// TIA Portal V20 export
ORGANIZATION_BLOCK "Main"   // OB1, LAD, ProgramCycle
TITLE = "Main Program Sweep (Cycle)"
{ S7_Optimized_Access := 'TRUE' }
// stored: SetENOAutomatically false
   VAR_INPUT
      Initial_Call : Bool;   // Initial call of this OB
      Remanence : Bool;   // =True, if remanent data are available
   END_VAR
BEGIN

REGION Network 1: SideShifter2
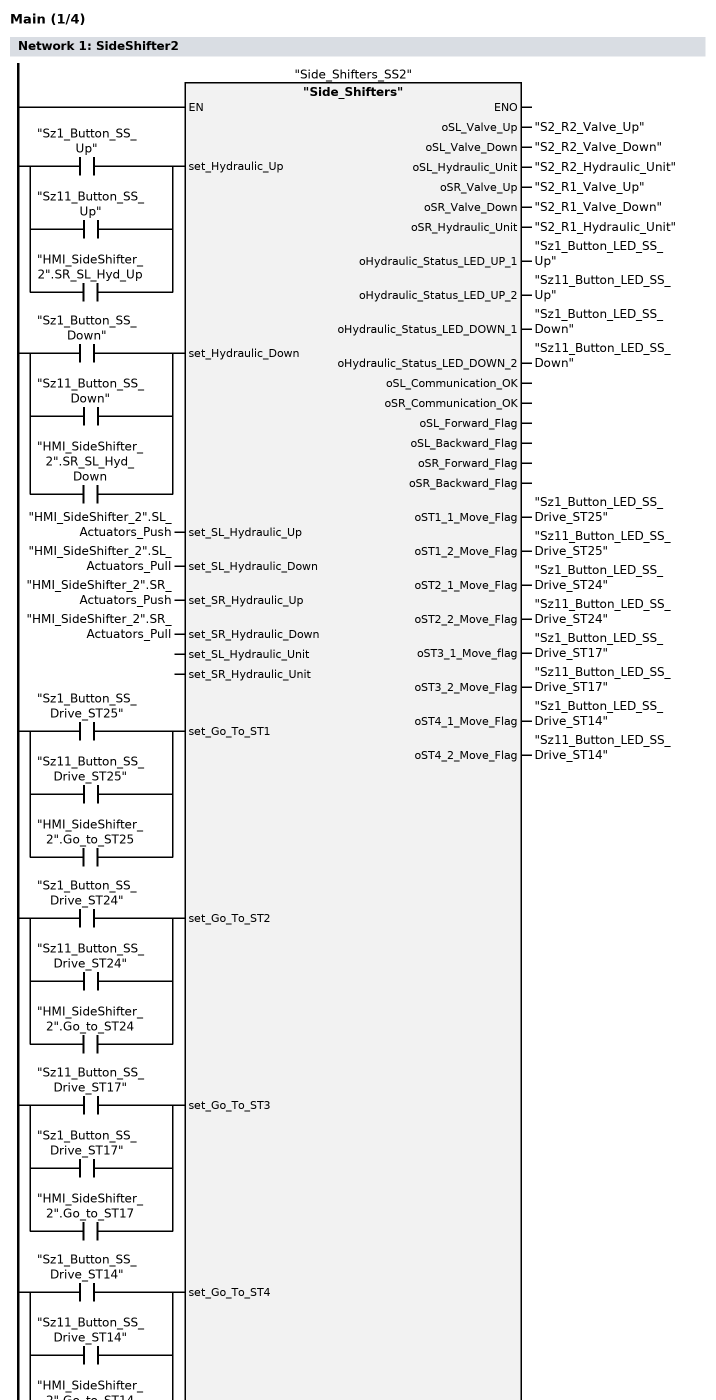
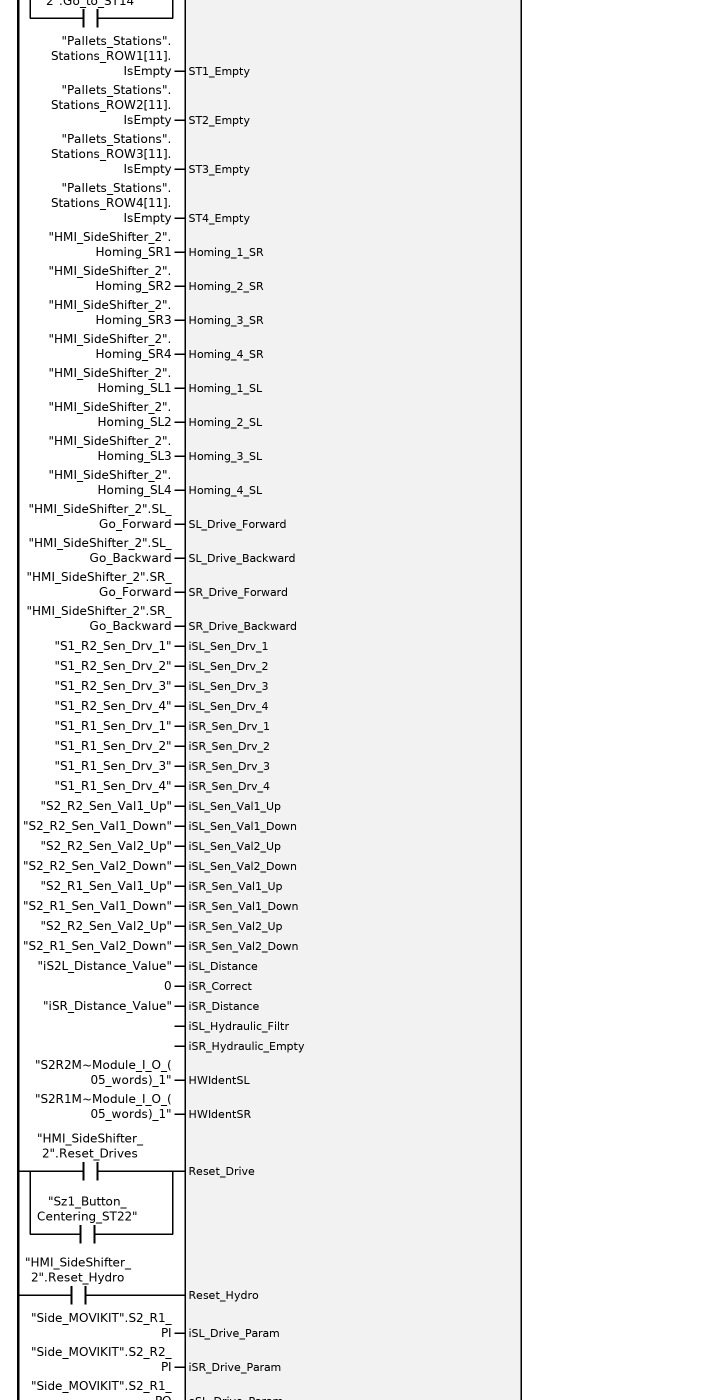
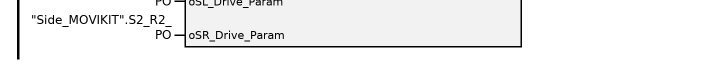
   RUNG wire#powerrail
      "Side_Shifters_SS2"(set_Hydraulic_Up := wire#w1, set_Hydraulic_Down := wire#w2, set_Go_To_ST1 := wire#w3, set_Go_To_ST2 := wire#w4, set_Go_To_ST3 := wire#w5, set_Go_To_ST4 := wire#w6, Reset_Drive := wire#w7, Reset_Hydro := wire#w8, set_SL_Hydraulic_Up := "HMI_SideShifter_2".SL_Actuators_Push, set_SL_Hydraulic_Down := "HMI_SideShifter_2".SL_Actuators_Pull, set_SR_Hydraulic_Up := "HMI_SideShifter_2".SR_Actuators_Push, set_SR_Hydraulic_Down := "HMI_SideShifter_2".SR_Actuators_Pull, set_SL_Hydraulic_Unit :=, set_SR_Hydraulic_Unit :=, ST1_Empty := "Pallets_Stations".Stations_ROW1[11].IsEmpty, ST2_Empty := "Pallets_Stations".Stations_ROW2[11].IsEmpty, ST3_Empty := "Pallets_Stations".Stations_ROW3[11].IsEmpty, ST4_Empty := "Pallets_Stations".Stations_ROW4[11].IsEmpty, Homing_1_SR := "HMI_SideShifter_2".Homing_SR1, Homing_2_SR := "HMI_SideShifter_2".Homing_SR2, Homing_3_SR := "HMI_SideShifter_2".Homing_SR3, Homing_4_SR := "HMI_SideShifter_2".Homing_SR4, Homing_1_SL := "HMI_SideShifter_2".Homing_SL1, Homing_2_SL := "HMI_SideShifter_2".Homing_SL2, Homing_3_SL := "HMI_SideShifter_2".Homing_SL3, Homing_4_SL := "HMI_SideShifter_2".Homing_SL4, SL_Drive_Forward := "HMI_SideShifter_2".SL_Go_Forward, SL_Drive_Backward := "HMI_SideShifter_2".SL_Go_Backward, SR_Drive_Forward := "HMI_SideShifter_2".SR_Go_Forward, SR_Drive_Backward := "HMI_SideShifter_2".SR_Go_Backward, iSL_Sen_Drv_1 := "S1_R2_Sen_Drv_1", iSL_Sen_Drv_2 := "S1_R2_Sen_Drv_2", iSL_Sen_Drv_3 := "S1_R2_Sen_Drv_3", iSL_Sen_Drv_4 := "S1_R2_Sen_Drv_4", iSR_Sen_Drv_1 := "S1_R1_Sen_Drv_1", iSR_Sen_Drv_2 := "S1_R1_Sen_Drv_2", iSR_Sen_Drv_3 := "S1_R1_Sen_Drv_3", iSR_Sen_Drv_4 := "S1_R1_Sen_Drv_4", iSL_Sen_Val1_Up := "S2_R2_Sen_Val1_Up", iSL_Sen_Val1_Down := "S2_R2_Sen_Val1_Down", iSL_Sen_Val2_Up := "S2_R2_Sen_Val2_Up", iSL_Sen_Val2_Down := "S2_R2_Sen_Val2_Down", iSR_Sen_Val1_Up := "S2_R1_Sen_Val1_Up", iSR_Sen_Val1_Down := "S2_R1_Sen_Val1_Down", iSR_Sen_Val2_Up := "S2_R2_Sen_Val2_Up", iSR_Sen_Val2_Down := "S2_R1_Sen_Val2_Down", iSL_Distance := "iS2L_Distance_Value", iSR_Correct := 0, iSR_Distance := "iSR_Distance_Value", iSL_Hydraulic_Filtr :=, iSR_Hydraulic_Empty :=, HWIdentSL := "S2R2M~Module_I_O_(05_words)_1", HWIdentSR := "S2R1M~Module_I_O_(05_words)_1", iSL_Drive_Param := "Side_MOVIKIT".S2_R1_PI, iSR_Drive_Param := "Side_MOVIKIT".S2_R2_PI, oSL_Drive_Param := "Side_MOVIKIT".S2_R1_PO, oSR_Drive_Param := "Side_MOVIKIT".S2_R2_PO, oSL_Valve_Up => "S2_R2_Valve_Up", oSL_Valve_Down => "S2_R2_Valve_Down", oSL_Hydraulic_Unit => "S2_R2_Hydraulic_Unit", oSR_Valve_Up => "S2_R1_Valve_Up", oSR_Valve_Down => "S2_R1_Valve_Down", oSR_Hydraulic_Unit => "S2_R1_Hydraulic_Unit", oHydraulic_Status_LED_UP_1 => "Sz1_Button_LED_SS_Up", oHydraulic_Status_LED_UP_2 => "Sz11_Button_LED_SS_Up", oHydraulic_Status_LED_DOWN_1 => "Sz1_Button_LED_SS_Down", oHydraulic_Status_LED_DOWN_2 => "Sz11_Button_LED_SS_Down", oSL_Communication_OK =>, oSR_Communication_OK =>, oSL_Forward_Flag =>, oSL_Backward_Flag =>, oSR_Forward_Flag =>, oSR_Backward_Flag =>, oST1_1_Move_Flag => "Sz1_Button_LED_SS_Drive_ST25", oST1_2_Move_Flag => "Sz11_Button_LED_SS_Drive_ST25", oST2_1_Move_Flag => "Sz1_Button_LED_SS_Drive_ST24", oST2_2_Move_Flag => "Sz11_Button_LED_SS_Drive_ST24", oST3_1_Move_flag => "Sz1_Button_LED_SS_Drive_ST17", oST3_2_Move_Flag => "Sz11_Button_LED_SS_Drive_ST17", oST4_1_Move_Flag => "Sz1_Button_LED_SS_Drive_ST14", oST4_2_Move_Flag => "Sz11_Button_LED_SS_Drive_ST14")
   END_RUNG
   RUNG wire#powerrail
      Contact( "Sz1_Button_SS_Up" )
   END_RUNG wire#w1
   RUNG wire#powerrail
      Contact( "Sz11_Button_SS_Up" )
   END_RUNG wire#w1
   RUNG wire#powerrail
      Contact( "HMI_SideShifter_2".SR_SL_Hyd_Up )
   END_RUNG wire#w1
   RUNG wire#powerrail
      Contact( "Sz1_Button_SS_Down" )
   END_RUNG wire#w2
   RUNG wire#powerrail
      Contact( "Sz11_Button_SS_Down" )
   END_RUNG wire#w2
   RUNG wire#powerrail
      Contact( "HMI_SideShifter_2".SR_SL_Hyd_Down )
   END_RUNG wire#w2
   RUNG wire#powerrail
      Contact( "Sz1_Button_SS_Drive_ST25" )
   END_RUNG wire#w3
   RUNG wire#powerrail
      Contact( "Sz11_Button_SS_Drive_ST25" )
   END_RUNG wire#w3
   RUNG wire#powerrail
      Contact( "HMI_SideShifter_2".Go_to_ST25 )
   END_RUNG wire#w3
   RUNG wire#powerrail
      Contact( "Sz1_Button_SS_Drive_ST24" )
   END_RUNG wire#w4
   RUNG wire#powerrail
      Contact( "Sz11_Button_SS_Drive_ST24" )
   END_RUNG wire#w4
   RUNG wire#powerrail
      Contact( "HMI_SideShifter_2".Go_to_ST24 )
   END_RUNG wire#w4
   RUNG wire#powerrail
      Contact( "Sz11_Button_SS_Drive_ST17" )
   END_RUNG wire#w5
   RUNG wire#powerrail
      Contact( "Sz1_Button_SS_Drive_ST17" )
   END_RUNG wire#w5
   RUNG wire#powerrail
      Contact( "HMI_SideShifter_2".Go_to_ST17 )
   END_RUNG wire#w5
   RUNG wire#powerrail
      Contact( "Sz1_Button_SS_Drive_ST14" )
   END_RUNG wire#w6
   RUNG wire#powerrail
      Contact( "Sz11_Button_SS_Drive_ST14" )
   END_RUNG wire#w6
   RUNG wire#powerrail
      Contact( "HMI_SideShifter_2".Go_to_ST14 )
   END_RUNG wire#w6
   RUNG wire#powerrail
      Contact( "HMI_SideShifter_2".Reset_Drives )
   END_RUNG wire#w7
   RUNG wire#powerrail
      Contact( "Sz1_Button_Centering_ST22" )
   END_RUNG wire#w7
   RUNG wire#powerrail
      Contact( "HMI_SideShifter_2".Reset_Hydro )
   END_RUNG wire#w8
   // the same network as SCL:
   "Side_Shifters_SS2"(set_Hydraulic_Up := "Sz1_Button_SS_Up" OR "Sz11_Button_SS_Up" OR "HMI_SideShifter_2".SR_SL_Hyd_Up,   // "Side_Shifters"
                       set_Hydraulic_Down := "Sz1_Button_SS_Down" OR "Sz11_Button_SS_Down" OR "HMI_SideShifter_2".SR_SL_Hyd_Down,
                       set_SL_Hydraulic_Up := "HMI_SideShifter_2".SL_Actuators_Push,
                       set_SL_Hydraulic_Down := "HMI_SideShifter_2".SL_Actuators_Pull,
                       set_SR_Hydraulic_Up := "HMI_SideShifter_2".SR_Actuators_Push,
                       set_SR_Hydraulic_Down := "HMI_SideShifter_2".SR_Actuators_Pull,
                       set_Go_To_ST1 := "Sz1_Button_SS_Drive_ST25" OR "Sz11_Button_SS_Drive_ST25" OR "HMI_SideShifter_2".Go_to_ST25,
                       set_Go_To_ST2 := "Sz1_Button_SS_Drive_ST24" OR "Sz11_Button_SS_Drive_ST24" OR "HMI_SideShifter_2".Go_to_ST24,
                       set_Go_To_ST3 := "Sz11_Button_SS_Drive_ST17" OR "Sz1_Button_SS_Drive_ST17" OR "HMI_SideShifter_2".Go_to_ST17,
                       set_Go_To_ST4 := "Sz1_Button_SS_Drive_ST14" OR "Sz11_Button_SS_Drive_ST14" OR "HMI_SideShifter_2".Go_to_ST14,
                       ST1_Empty := "Pallets_Stations".Stations_ROW1[11].IsEmpty,
                       ST2_Empty := "Pallets_Stations".Stations_ROW2[11].IsEmpty,
                       ST3_Empty := "Pallets_Stations".Stations_ROW3[11].IsEmpty,
                       ST4_Empty := "Pallets_Stations".Stations_ROW4[11].IsEmpty,
                       Homing_1_SR := "HMI_SideShifter_2".Homing_SR1,
                       Homing_2_SR := "HMI_SideShifter_2".Homing_SR2,
                       Homing_3_SR := "HMI_SideShifter_2".Homing_SR3,
                       Homing_4_SR := "HMI_SideShifter_2".Homing_SR4,
                       Homing_1_SL := "HMI_SideShifter_2".Homing_SL1,
                       Homing_2_SL := "HMI_SideShifter_2".Homing_SL2,
                       Homing_3_SL := "HMI_SideShifter_2".Homing_SL3,
                       Homing_4_SL := "HMI_SideShifter_2".Homing_SL4,
                       SL_Drive_Forward := "HMI_SideShifter_2".SL_Go_Forward,
                       SL_Drive_Backward := "HMI_SideShifter_2".SL_Go_Backward,
                       SR_Drive_Forward := "HMI_SideShifter_2".SR_Go_Forward,
                       SR_Drive_Backward := "HMI_SideShifter_2".SR_Go_Backward,
                       iSL_Sen_Drv_1 := "S1_R2_Sen_Drv_1",
                       iSL_Sen_Drv_2 := "S1_R2_Sen_Drv_2",
                       iSL_Sen_Drv_3 := "S1_R2_Sen_Drv_3",
                       iSL_Sen_Drv_4 := "S1_R2_Sen_Drv_4",
                       iSR_Sen_Drv_1 := "S1_R1_Sen_Drv_1",
                       iSR_Sen_Drv_2 := "S1_R1_Sen_Drv_2",
                       iSR_Sen_Drv_3 := "S1_R1_Sen_Drv_3",
                       iSR_Sen_Drv_4 := "S1_R1_Sen_Drv_4",
                       iSL_Sen_Val1_Up := "S2_R2_Sen_Val1_Up",
                       iSL_Sen_Val1_Down := "S2_R2_Sen_Val1_Down",
                       iSL_Sen_Val2_Up := "S2_R2_Sen_Val2_Up",
                       iSL_Sen_Val2_Down := "S2_R2_Sen_Val2_Down",
                       iSR_Sen_Val1_Up := "S2_R1_Sen_Val1_Up",
                       iSR_Sen_Val1_Down := "S2_R1_Sen_Val1_Down",
                       iSR_Sen_Val2_Up := "S2_R2_Sen_Val2_Up",
                       iSR_Sen_Val2_Down := "S2_R1_Sen_Val2_Down",
                       iSL_Distance := "iS2L_Distance_Value",
                       iSR_Correct := 0,
                       iSR_Distance := "iSR_Distance_Value",
                       HWIdentSL := "S2R2M~Module_I_O_(05_words)_1",
                       HWIdentSR := "S2R1M~Module_I_O_(05_words)_1",
                       Reset_Drive := "HMI_SideShifter_2".Reset_Drives OR "Sz1_Button_Centering_ST22",
                       Reset_Hydro := "HMI_SideShifter_2".Reset_Hydro,
                       iSL_Drive_Param := "Side_MOVIKIT".S2_R1_PI,
                       iSR_Drive_Param := "Side_MOVIKIT".S2_R2_PI,
                       oSL_Drive_Param := "Side_MOVIKIT".S2_R1_PO,
                       oSR_Drive_Param := "Side_MOVIKIT".S2_R2_PO,
                       oSL_Valve_Up => "S2_R2_Valve_Up",
                       oSL_Valve_Down => "S2_R2_Valve_Down",
                       oSL_Hydraulic_Unit => "S2_R2_Hydraulic_Unit",
                       oSR_Valve_Up => "S2_R1_Valve_Up",
                       oSR_Valve_Down => "S2_R1_Valve_Down",
                       oSR_Hydraulic_Unit => "S2_R1_Hydraulic_Unit",
                       oHydraulic_Status_LED_UP_1 => "Sz1_Button_LED_SS_Up",
                       oHydraulic_Status_LED_UP_2 => "Sz11_Button_LED_SS_Up",
                       oHydraulic_Status_LED_DOWN_1 => "Sz1_Button_LED_SS_Down",
                       oHydraulic_Status_LED_DOWN_2 => "Sz11_Button_LED_SS_Down",
                       oST1_1_Move_Flag => "Sz1_Button_LED_SS_Drive_ST25",
                       oST1_2_Move_Flag => "Sz11_Button_LED_SS_Drive_ST25",
                       oST2_1_Move_Flag => "Sz1_Button_LED_SS_Drive_ST24",
                       oST2_2_Move_Flag => "Sz11_Button_LED_SS_Drive_ST24",
                       oST3_1_Move_flag => "Sz1_Button_LED_SS_Drive_ST17",
                       oST3_2_Move_Flag => "Sz11_Button_LED_SS_Drive_ST17",
                       oST4_1_Move_Flag => "Sz1_Button_LED_SS_Drive_ST14",
                       oST4_2_Move_Flag => "Sz11_Button_LED_SS_Drive_ST14");
END_REGION

REGION Network 2: SideShifter 1
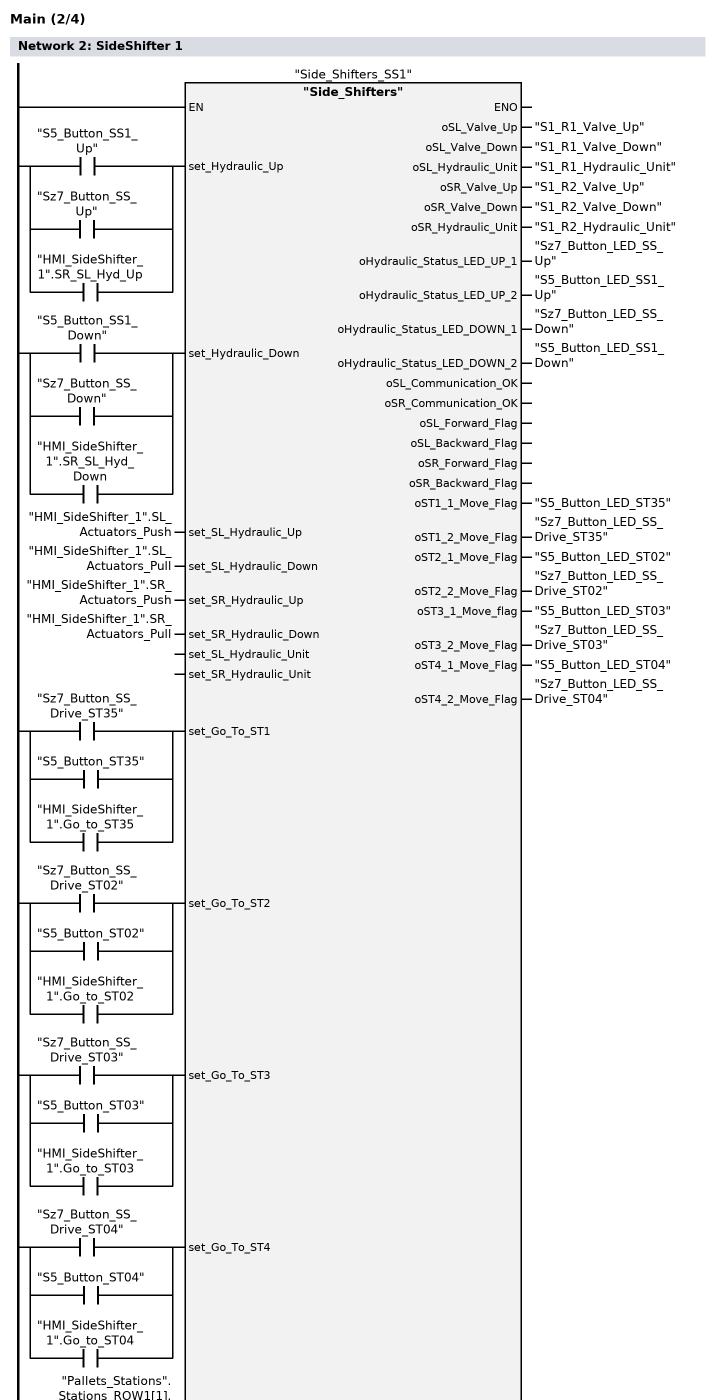
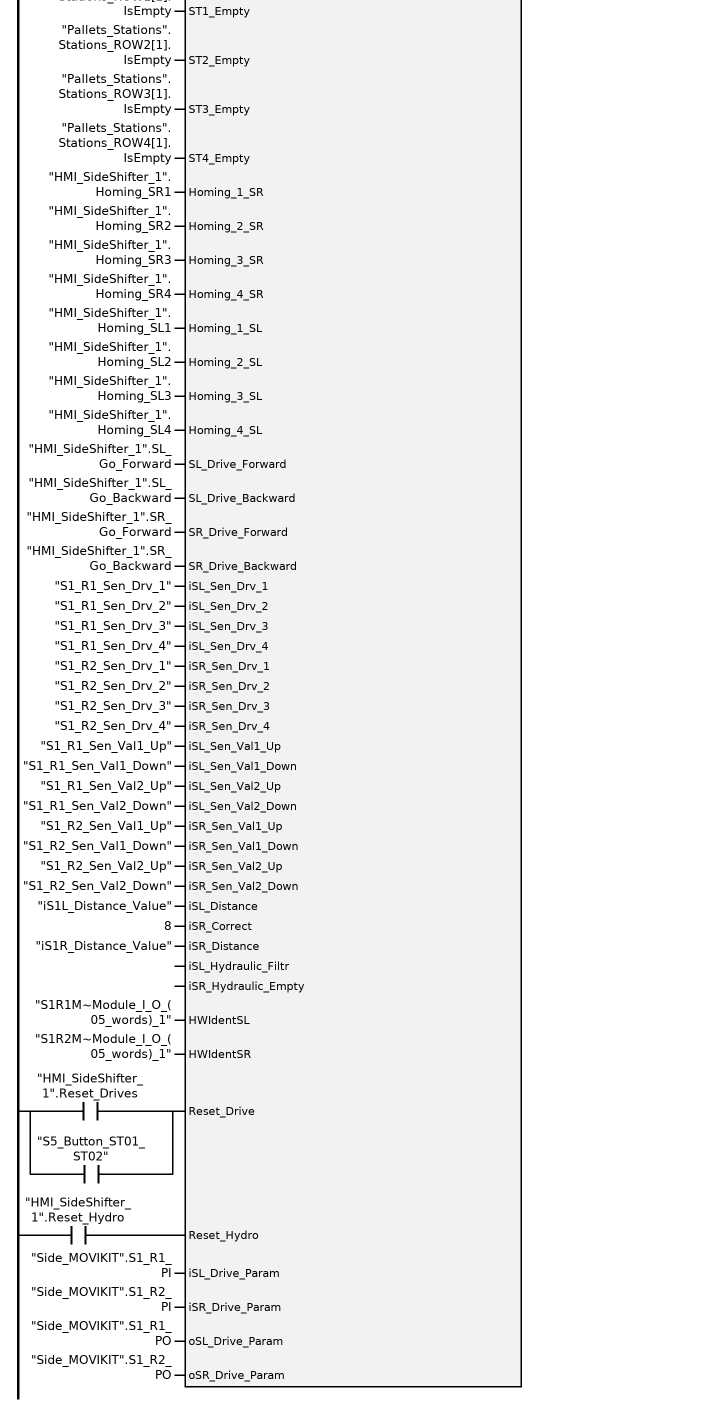
   RUNG wire#powerrail
      "Side_Shifters_SS1"(set_Hydraulic_Up := wire#w1, set_Hydraulic_Down := wire#w2, set_Go_To_ST1 := wire#w3, set_Go_To_ST2 := wire#w4, set_Go_To_ST3 := wire#w5, set_Go_To_ST4 := wire#w6, Reset_Drive := wire#w7, Reset_Hydro := wire#w8, set_SL_Hydraulic_Up := "HMI_SideShifter_1".SL_Actuators_Push, set_SL_Hydraulic_Down := "HMI_SideShifter_1".SL_Actuators_Pull, set_SR_Hydraulic_Up := "HMI_SideShifter_1".SR_Actuators_Push, set_SR_Hydraulic_Down := "HMI_SideShifter_1".SR_Actuators_Pull, set_SL_Hydraulic_Unit :=, set_SR_Hydraulic_Unit :=, ST1_Empty := "Pallets_Stations".Stations_ROW1[1].IsEmpty, ST2_Empty := "Pallets_Stations".Stations_ROW2[1].IsEmpty, ST3_Empty := "Pallets_Stations".Stations_ROW3[1].IsEmpty, ST4_Empty := "Pallets_Stations".Stations_ROW4[1].IsEmpty, Homing_1_SR := "HMI_SideShifter_1".Homing_SR1, Homing_2_SR := "HMI_SideShifter_1".Homing_SR2, Homing_3_SR := "HMI_SideShifter_1".Homing_SR3, Homing_4_SR := "HMI_SideShifter_1".Homing_SR4, Homing_1_SL := "HMI_SideShifter_1".Homing_SL1, Homing_2_SL := "HMI_SideShifter_1".Homing_SL2, Homing_3_SL := "HMI_SideShifter_1".Homing_SL3, Homing_4_SL := "HMI_SideShifter_1".Homing_SL4, SL_Drive_Forward := "HMI_SideShifter_1".SL_Go_Forward, SL_Drive_Backward := "HMI_SideShifter_1".SL_Go_Backward, SR_Drive_Forward := "HMI_SideShifter_1".SR_Go_Forward, SR_Drive_Backward := "HMI_SideShifter_1".SR_Go_Backward, iSL_Sen_Drv_1 := "S1_R1_Sen_Drv_1", iSL_Sen_Drv_2 := "S1_R1_Sen_Drv_2", iSL_Sen_Drv_3 := "S1_R1_Sen_Drv_3", iSL_Sen_Drv_4 := "S1_R1_Sen_Drv_4", iSR_Sen_Drv_1 := "S1_R2_Sen_Drv_1", iSR_Sen_Drv_2 := "S1_R2_Sen_Drv_2", iSR_Sen_Drv_3 := "S1_R2_Sen_Drv_3", iSR_Sen_Drv_4 := "S1_R2_Sen_Drv_4", iSL_Sen_Val1_Up := "S1_R1_Sen_Val1_Up", iSL_Sen_Val1_Down := "S1_R1_Sen_Val1_Down", iSL_Sen_Val2_Up := "S1_R1_Sen_Val2_Up", iSL_Sen_Val2_Down := "S1_R1_Sen_Val2_Down", iSR_Sen_Val1_Up := "S1_R2_Sen_Val1_Up", iSR_Sen_Val1_Down := "S1_R2_Sen_Val1_Down", iSR_Sen_Val2_Up := "S1_R2_Sen_Val2_Up", iSR_Sen_Val2_Down := "S1_R2_Sen_Val2_Down", iSL_Distance := "iS1L_Distance_Value", iSR_Correct := 8, iSR_Distance := "iS1R_Distance_Value", iSL_Hydraulic_Filtr :=, iSR_Hydraulic_Empty :=, HWIdentSL := "S1R1M~Module_I_O_(05_words)_1", HWIdentSR := "S1R2M~Module_I_O_(05_words)_1", iSL_Drive_Param := "Side_MOVIKIT".S1_R1_PI, iSR_Drive_Param := "Side_MOVIKIT".S1_R2_PI, oSL_Drive_Param := "Side_MOVIKIT".S1_R1_PO, oSR_Drive_Param := "Side_MOVIKIT".S1_R2_PO, oSL_Valve_Up => "S1_R1_Valve_Up", oSL_Valve_Down => "S1_R1_Valve_Down", oSL_Hydraulic_Unit => "S1_R1_Hydraulic_Unit", oSR_Valve_Up => "S1_R2_Valve_Up", oSR_Valve_Down => "S1_R2_Valve_Down", oSR_Hydraulic_Unit => "S1_R2_Hydraulic_Unit", oHydraulic_Status_LED_UP_1 => "Sz7_Button_LED_SS_Up", oHydraulic_Status_LED_UP_2 => "S5_Button_LED_SS1_Up", oHydraulic_Status_LED_DOWN_1 => "Sz7_Button_LED_SS_Down", oHydraulic_Status_LED_DOWN_2 => "S5_Button_LED_SS1_Down", oSL_Communication_OK =>, oSR_Communication_OK =>, oSL_Forward_Flag =>, oSL_Backward_Flag =>, oSR_Forward_Flag =>, oSR_Backward_Flag =>, oST1_1_Move_Flag => "S5_Button_LED_ST35", oST1_2_Move_Flag => "Sz7_Button_LED_SS_Drive_ST35", oST2_1_Move_Flag => "S5_Button_LED_ST02", oST2_2_Move_Flag => "Sz7_Button_LED_SS_Drive_ST02", oST3_1_Move_flag => "S5_Button_LED_ST03", oST3_2_Move_Flag => "Sz7_Button_LED_SS_Drive_ST03", oST4_1_Move_Flag => "S5_Button_LED_ST04", oST4_2_Move_Flag => "Sz7_Button_LED_SS_Drive_ST04")
   END_RUNG
   RUNG wire#powerrail
      Contact( "S5_Button_SS1_Up" )
   END_RUNG wire#w1
   RUNG wire#powerrail
      Contact( "Sz7_Button_SS_Up" )
   END_RUNG wire#w1
   RUNG wire#powerrail
      Contact( "HMI_SideShifter_1".SR_SL_Hyd_Up )
   END_RUNG wire#w1
   RUNG wire#powerrail
      Contact( "S5_Button_SS1_Down" )
   END_RUNG wire#w2
   RUNG wire#powerrail
      Contact( "Sz7_Button_SS_Down" )
   END_RUNG wire#w2
   RUNG wire#powerrail
      Contact( "HMI_SideShifter_1".SR_SL_Hyd_Down )
   END_RUNG wire#w2
   RUNG wire#powerrail
      Contact( "Sz7_Button_SS_Drive_ST35" )
   END_RUNG wire#w3
   RUNG wire#powerrail
      Contact( "S5_Button_ST35" )
   END_RUNG wire#w3
   RUNG wire#powerrail
      Contact( "HMI_SideShifter_1".Go_to_ST35 )
   END_RUNG wire#w3
   RUNG wire#powerrail
      Contact( "Sz7_Button_SS_Drive_ST02" )
   END_RUNG wire#w4
   RUNG wire#powerrail
      Contact( "S5_Button_ST02" )
   END_RUNG wire#w4
   RUNG wire#powerrail
      Contact( "HMI_SideShifter_1".Go_to_ST02 )
   END_RUNG wire#w4
   RUNG wire#powerrail
      Contact( "Sz7_Button_SS_Drive_ST03" )
   END_RUNG wire#w5
   RUNG wire#powerrail
      Contact( "S5_Button_ST03" )
   END_RUNG wire#w5
   RUNG wire#powerrail
      Contact( "HMI_SideShifter_1".Go_to_ST03 )
   END_RUNG wire#w5
   RUNG wire#powerrail
      Contact( "Sz7_Button_SS_Drive_ST04" )
   END_RUNG wire#w6
   RUNG wire#powerrail
      Contact( "S5_Button_ST04" )
   END_RUNG wire#w6
   RUNG wire#powerrail
      Contact( "HMI_SideShifter_1".Go_to_ST04 )
   END_RUNG wire#w6
   RUNG wire#powerrail
      Contact( "HMI_SideShifter_1".Reset_Drives )
   END_RUNG wire#w7
   RUNG wire#powerrail
      Contact( "S5_Button_ST01_ST02" )
   END_RUNG wire#w7
   RUNG wire#powerrail
      Contact( "HMI_SideShifter_1".Reset_Hydro )
   END_RUNG wire#w8
   // the same network as SCL:
   "Side_Shifters_SS1"(set_Hydraulic_Up := "S5_Button_SS1_Up" OR "Sz7_Button_SS_Up" OR "HMI_SideShifter_1".SR_SL_Hyd_Up,   // "Side_Shifters"
                       set_Hydraulic_Down := "S5_Button_SS1_Down" OR "Sz7_Button_SS_Down" OR "HMI_SideShifter_1".SR_SL_Hyd_Down,
                       set_SL_Hydraulic_Up := "HMI_SideShifter_1".SL_Actuators_Push,
                       set_SL_Hydraulic_Down := "HMI_SideShifter_1".SL_Actuators_Pull,
                       set_SR_Hydraulic_Up := "HMI_SideShifter_1".SR_Actuators_Push,
                       set_SR_Hydraulic_Down := "HMI_SideShifter_1".SR_Actuators_Pull,
                       set_Go_To_ST1 := "Sz7_Button_SS_Drive_ST35" OR "S5_Button_ST35" OR "HMI_SideShifter_1".Go_to_ST35,
                       set_Go_To_ST2 := "Sz7_Button_SS_Drive_ST02" OR "S5_Button_ST02" OR "HMI_SideShifter_1".Go_to_ST02,
                       set_Go_To_ST3 := "Sz7_Button_SS_Drive_ST03" OR "S5_Button_ST03" OR "HMI_SideShifter_1".Go_to_ST03,
                       set_Go_To_ST4 := "Sz7_Button_SS_Drive_ST04" OR "S5_Button_ST04" OR "HMI_SideShifter_1".Go_to_ST04,
                       ST1_Empty := "Pallets_Stations".Stations_ROW1[1].IsEmpty,
                       ST2_Empty := "Pallets_Stations".Stations_ROW2[1].IsEmpty,
                       ST3_Empty := "Pallets_Stations".Stations_ROW3[1].IsEmpty,
                       ST4_Empty := "Pallets_Stations".Stations_ROW4[1].IsEmpty,
                       Homing_1_SR := "HMI_SideShifter_1".Homing_SR1,
                       Homing_2_SR := "HMI_SideShifter_1".Homing_SR2,
                       Homing_3_SR := "HMI_SideShifter_1".Homing_SR3,
                       Homing_4_SR := "HMI_SideShifter_1".Homing_SR4,
                       Homing_1_SL := "HMI_SideShifter_1".Homing_SL1,
                       Homing_2_SL := "HMI_SideShifter_1".Homing_SL2,
                       Homing_3_SL := "HMI_SideShifter_1".Homing_SL3,
                       Homing_4_SL := "HMI_SideShifter_1".Homing_SL4,
                       SL_Drive_Forward := "HMI_SideShifter_1".SL_Go_Forward,
                       SL_Drive_Backward := "HMI_SideShifter_1".SL_Go_Backward,
                       SR_Drive_Forward := "HMI_SideShifter_1".SR_Go_Forward,
                       SR_Drive_Backward := "HMI_SideShifter_1".SR_Go_Backward,
                       iSL_Sen_Drv_1 := "S1_R1_Sen_Drv_1",
                       iSL_Sen_Drv_2 := "S1_R1_Sen_Drv_2",
                       iSL_Sen_Drv_3 := "S1_R1_Sen_Drv_3",
                       iSL_Sen_Drv_4 := "S1_R1_Sen_Drv_4",
                       iSR_Sen_Drv_1 := "S1_R2_Sen_Drv_1",
                       iSR_Sen_Drv_2 := "S1_R2_Sen_Drv_2",
                       iSR_Sen_Drv_3 := "S1_R2_Sen_Drv_3",
                       iSR_Sen_Drv_4 := "S1_R2_Sen_Drv_4",
                       iSL_Sen_Val1_Up := "S1_R1_Sen_Val1_Up",
                       iSL_Sen_Val1_Down := "S1_R1_Sen_Val1_Down",
                       iSL_Sen_Val2_Up := "S1_R1_Sen_Val2_Up",
                       iSL_Sen_Val2_Down := "S1_R1_Sen_Val2_Down",
                       iSR_Sen_Val1_Up := "S1_R2_Sen_Val1_Up",
                       iSR_Sen_Val1_Down := "S1_R2_Sen_Val1_Down",
                       iSR_Sen_Val2_Up := "S1_R2_Sen_Val2_Up",
                       iSR_Sen_Val2_Down := "S1_R2_Sen_Val2_Down",
                       iSL_Distance := "iS1L_Distance_Value",
                       iSR_Correct := 8,
                       iSR_Distance := "iS1R_Distance_Value",
                       HWIdentSL := "S1R1M~Module_I_O_(05_words)_1",
                       HWIdentSR := "S1R2M~Module_I_O_(05_words)_1",
                       Reset_Drive := "HMI_SideShifter_1".Reset_Drives OR "S5_Button_ST01_ST02",
                       Reset_Hydro := "HMI_SideShifter_1".Reset_Hydro,
                       iSL_Drive_Param := "Side_MOVIKIT".S1_R1_PI,
                       iSR_Drive_Param := "Side_MOVIKIT".S1_R2_PI,
                       oSL_Drive_Param := "Side_MOVIKIT".S1_R1_PO,
                       oSR_Drive_Param := "Side_MOVIKIT".S1_R2_PO,
                       oSL_Valve_Up => "S1_R1_Valve_Up",
                       oSL_Valve_Down => "S1_R1_Valve_Down",
                       oSL_Hydraulic_Unit => "S1_R1_Hydraulic_Unit",
                       oSR_Valve_Up => "S1_R2_Valve_Up",
                       oSR_Valve_Down => "S1_R2_Valve_Down",
                       oSR_Hydraulic_Unit => "S1_R2_Hydraulic_Unit",
                       oHydraulic_Status_LED_UP_1 => "Sz7_Button_LED_SS_Up",
                       oHydraulic_Status_LED_UP_2 => "S5_Button_LED_SS1_Up",
                       oHydraulic_Status_LED_DOWN_1 => "Sz7_Button_LED_SS_Down",
                       oHydraulic_Status_LED_DOWN_2 => "S5_Button_LED_SS1_Down",
                       oST1_1_Move_Flag => "S5_Button_LED_ST35",
                       oST1_2_Move_Flag => "Sz7_Button_LED_SS_Drive_ST35",
                       oST2_1_Move_Flag => "S5_Button_LED_ST02",
                       oST2_2_Move_Flag => "Sz7_Button_LED_SS_Drive_ST02",
                       oST3_1_Move_flag => "S5_Button_LED_ST03",
                       oST3_2_Move_Flag => "Sz7_Button_LED_SS_Drive_ST03",
                       oST4_1_Move_Flag => "S5_Button_LED_ST04",
                       oST4_2_Move_Flag => "Sz7_Button_LED_SS_Drive_ST04");
END_REGION

REGION Network 3: Pallet Circulation
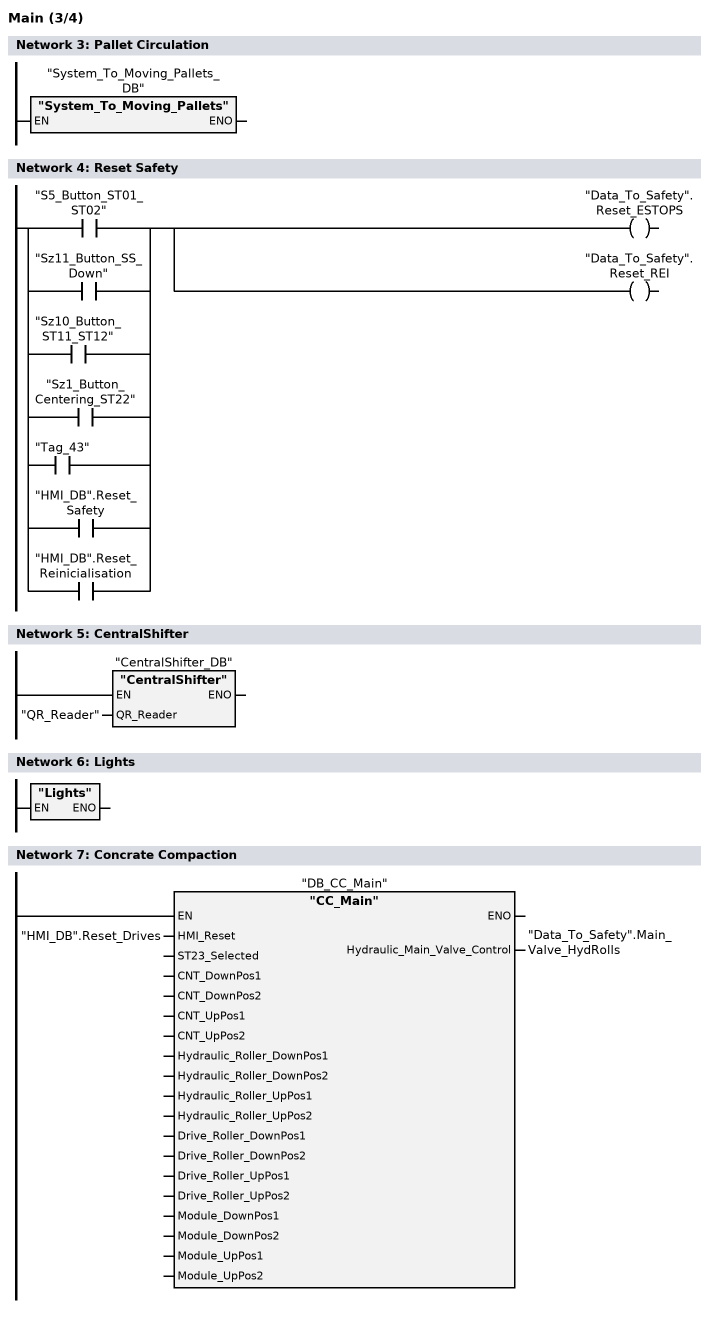
   RUNG wire#powerrail
      "System_To_Moving_Pallets_DB"()
   END_RUNG
   // the same network as SCL:
   "System_To_Moving_Pallets_DB"();   // "System_To_Moving_Pallets"
END_REGION

REGION Network 4: Reset Safety
   RUNG wire#powerrail
      Contact( "S5_Button_ST01_ST02" )
      wire#w1
      Coil( "Data_To_Safety".Reset_ESTOPS )
   END_RUNG
   RUNG wire#powerrail
      Contact( "Sz11_Button_SS_Down" )
   END_RUNG wire#w1
   RUNG wire#powerrail
      Contact( "Sz10_Button_ST11_ST12" )
   END_RUNG wire#w1
   RUNG wire#powerrail
      Contact( "Sz1_Button_Centering_ST22" )
   END_RUNG wire#w1
   RUNG wire#powerrail
      Contact( "Tag_43" )
   END_RUNG wire#w1
   RUNG wire#powerrail
      Contact( "HMI_DB".Reset_Safety )
   END_RUNG wire#w1
   RUNG wire#powerrail
      Contact( "HMI_DB".Reset_Reinicialisation )
   END_RUNG wire#w1
   RUNG wire#w1
      Coil( "Data_To_Safety".Reset_REI )
   END_RUNG
   // the same network as SCL:
   "Data_To_Safety".Reset_ESTOPS := "S5_Button_ST01_ST02" OR "Sz11_Button_SS_Down" OR "Sz10_Button_ST11_ST12" OR "Sz1_Button_Centering_ST22" OR "Tag_43" OR "HMI_DB".Reset_Safety OR "HMI_DB".Reset_Reinicialisation;
   "Data_To_Safety".Reset_REI := "Data_To_Safety".Reset_ESTOPS;
END_REGION

REGION Network 5: CentralShifter
   RUNG wire#powerrail
      "CentralShifter_DB"(QR_Reader := "QR_Reader")
   END_RUNG
   // the same network as SCL:
   "CentralShifter_DB"(QR_Reader := "QR_Reader");   // "CentralShifter"
END_REGION

REGION Network 6: Lights
   RUNG wire#powerrail
      "Lights"()
   END_RUNG
   // the same network as SCL:
   "Lights"();
END_REGION

REGION Network 7: Concrate Compaction
   RUNG wire#powerrail
      "DB_CC_Main"(HMI_Reset := "HMI_DB".Reset_Drives, ST23_Selected :=, CNT_DownPos1 :=, CNT_DownPos2 :=, CNT_UpPos1 :=, CNT_UpPos2 :=, Hydraulic_Roller_DownPos1 :=, Hydraulic_Roller_DownPos2 :=, Hydraulic_Roller_UpPos1 :=, Hydraulic_Roller_UpPos2 :=, Drive_Roller_DownPos1 :=, Drive_Roller_DownPos2 :=, Drive_Roller_UpPos1 :=, Drive_Roller_UpPos2 :=, Module_DownPos1 :=, Module_DownPos2 :=, Module_UpPos1 :=, Module_UpPos2 :=, Hydraulic_Main_Valve_Control => "Data_To_Safety".Main_Valve_HydRolls)
   END_RUNG
   // the same network as SCL:
   "DB_CC_Main"(HMI_Reset := "HMI_DB".Reset_Drives,   // "CC_Main"
                Hydraulic_Main_Valve_Control => "Data_To_Safety".Main_Valve_HydRolls);
END_REGION

REGION Network 8: Oil
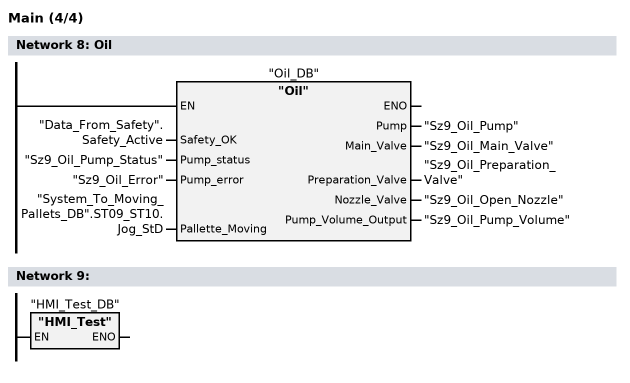
   RUNG wire#powerrail
      "Oil_DB"(Safety_OK := "Data_From_Safety".Safety_Active, Pump_status := "Sz9_Oil_Pump_Status", Pump_error := "Sz9_Oil_Error", Pallette_Moving := "System_To_Moving_Pallets_DB".ST09_ST10.Jog_StD, Pump => "Sz9_Oil_Pump", Main_Valve => "Sz9_Oil_Main_Valve", Preparation_Valve => "Sz9_Oil_Preparation_Valve", Nozzle_Valve => "Sz9_Oil_Open_Nozzle", Pump_Volume_Output => "Sz9_Oil_Pump_Volume")
   END_RUNG
   // the same network as SCL:
   "Oil_DB"(Safety_OK := "Data_From_Safety".Safety_Active,   // "Oil"
            Pump_status := "Sz9_Oil_Pump_Status",
            Pump_error := "Sz9_Oil_Error",
            Pallette_Moving := "System_To_Moving_Pallets_DB".ST09_ST10.Jog_StD,
            Pump => "Sz9_Oil_Pump",
            Main_Valve => "Sz9_Oil_Main_Valve",
            Preparation_Valve => "Sz9_Oil_Preparation_Valve",
            Nozzle_Valve => "Sz9_Oil_Open_Nozzle",
            Pump_Volume_Output => "Sz9_Oil_Pump_Volume");
END_REGION

REGION Network 9
   RUNG wire#powerrail
      "HMI_Test_DB"()
   END_RUNG
   // the same network as SCL:
   "HMI_Test_DB"();   // "HMI_Test"
END_REGION
END_ORGANIZATION_BLOCK
